FUNCTION_BLOCK ABSTRACT Spline
VAR_INPUT
END_VAR
VAR_OUTPUT
END_VAR
VAR
	lengthVar     :LREAL;
	startPoint 	  : RobotPoseSimple;
	endPoint      : RobotPoseSimple;
END_VAR

METHOD PROTECTED ABSTRACT calculateLength : LREAL
VAR_INPUT
END_VAR
END_METHOD

METHOD ABSTRACT diff : RobotPoseSimple
VAR_INPUT
	arcLength: LREAL;
	order: INT := 1;
END_VAR
END_METHOD

PROPERTY endPointVal : RobotPoseSimple
GET
endPointVal := endPoint;
END_GET
SET
END_SET
END_PROPERTY

METHOD PUBLIC ABSTRACT getPoint : RobotPoseSimple
VAR_INPUT
	arcLength: LREAL;
END_VAR
END_METHOD

PROPERTY length : LREAL
GET
 length := lengthVar;
END_GET
SET
END_SET
END_PROPERTY

PROPERTY startPointVal : RobotPoseSimple
GET
startPointVal.x := startPoint.x;
startPointVal.y := startPoint.y;
startPointVal.theta := startPoint.theta;
END_GET
SET
END_SET
END_PROPERTY

END_FUNCTION_BLOCK

(* stored: Version 1.1.0.1, ProductVersion 3.1.4024.11
   POU Spline: Id {962108ba-b764-4703-887f-44bc4cb4c5ee}, SpecialFunc None
   Method calculateLength: Id {4c02d6a5-f067-4f4f-86c9-78561224f2c0}
   Method diff: Id {abb1aec0-c192-43c2-a1a2-b654a47047f5}
   Property endPointVal: Id {7962ae8b-69b1-4349-8d50-e8cc4dc9821e}
   Get Get: Id {874295b2-4f0f-444d-8da3-65f51689f278}
   Set Set: Id {0a3c1837-43da-4af9-9891-48210de97902}
   Method getPoint: Id {e1cf1b15-c371-4375-8f5b-cd02de7ff7af}
   Property length: Id {8ff29e3f-4d60-4193-9ab3-f3fd25f3230c}
   Get Get: Id {4402e7a9-338c-477a-a725-7a816516dece}
   Set Set: Id {28a4e29e-362e-4b36-b064-686c9255d71b}
   Property startPointVal: Id {31816552-8dd4-4368-92f9-6cd8ac4228ea}
   Get Get: Id {a5ae9440-f337-4737-a62f-30ed86d8e10f}
   Set Set: Id {9518b61d-5289-4168-b250-5ef7f6373079} *)
